PROGRAM MAIN
VAR
	//cmt 1
	bTest_1 : BOOL;
	bThuc: BOOL;
	bThuc2: BOOL;
END_VAR

END_PROGRAM

(* stored: Version 1.1.0.1, ProductVersion 3.1.4024.11
   POU MAIN: Id {0901d40b-d0af-40a4-bd60-64fc45002868}, SpecialFunc None *)
